(* PLC project Unnamed, Unknown Unnamed 1 *)
(* stored: creationDateTime 2022-02-07T10:15:24, modificationDateTime 2022-04-01T00:18:43 *)

PROGRAM program0
  VAR
    IN0 : BOOL;
    IN1 : BOOL;
    IN2 : BOOL;
    OUT : BOOL;
  END_VAR

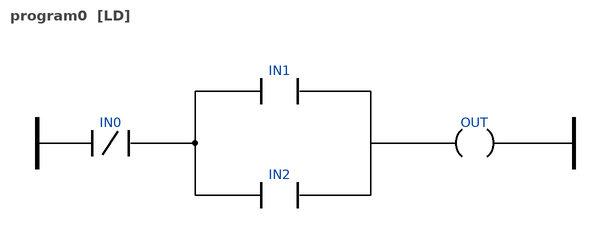
(* LD diagram, written out as Structured Text *)
OUT := NOT IN0 AND (IN1 OR IN2);
END_PROGRAM

CONFIGURATION Config0
  RESOURCE Res0 ON PLC
    TASK task0(INTERVAL := T#20ms, PRIORITY := 0);
    PROGRAM instance0 WITH task0 : program0;
  END_RESOURCE
END_CONFIGURATION
